// TIA Portal V20 export
DATA_BLOCK "zPTPMC_Data"   // DB362
// stored: MemoryReserve 100, Namespace CITI_Logic
   VAR
      PTPMC_Data : Array[0..29] of "CITI_Logic.zp_CITIData";
      CheckSum { S7_SetPoint := 'True'} : Array[1..16] of DWord;
   END_VAR
BEGIN
END_DATA_BLOCK
